FUNCTION_BLOCK FB_System_KKKW_145
VAR_INPUT

	Freigabe_auto			: BOOL;
	Freigabe_Deakt_auto		: BOOL;
	Betrieb_Anford_auto		: BOOL;

	Regelung_Modus_auto		: SINT;
	Regelung_Sollw_auto		: REAL;
END_VAR
VAR_OUTPUT
	{attribute 'OPC.UA.DA' := '1'}Parameter		: ST_System_KKKW_Parameter;   
	{attribute 'OPC.UA.DA' := '1'}Zustand			: ST_System_KKKW_Zustand;	
	{attribute 'OPC.UA.DA' := '1'}Stellwert		: ST_System_KKKW_Stellwert;  	
	{attribute 'OPC.UA.DA' := '1'}Steuerung		: ST_System_KKKW_Steuerung;  	
END_VAR
VAR
	Pumpe_145		: FB_PU;
	Stellventil_145	: FB_SV;
	Ablaufsteuerung	: FB_System_KKKW_Ablaufsteuerung;
	Logik			: FB_System_KKKW_Logik;
	Zustandscheck	: FB_System_KKKW_Zustandscheck;
	Stellwertscheck	: FB_System_KKKW_Stellwertscheck;
	Sollwertscheck	: FB_System_KKKW_Sollwertscheck;
END_VAR
VAR // added by the converter: edge detectors and wires of the graphical bodies
    _w1 : ANY;
END_VAR

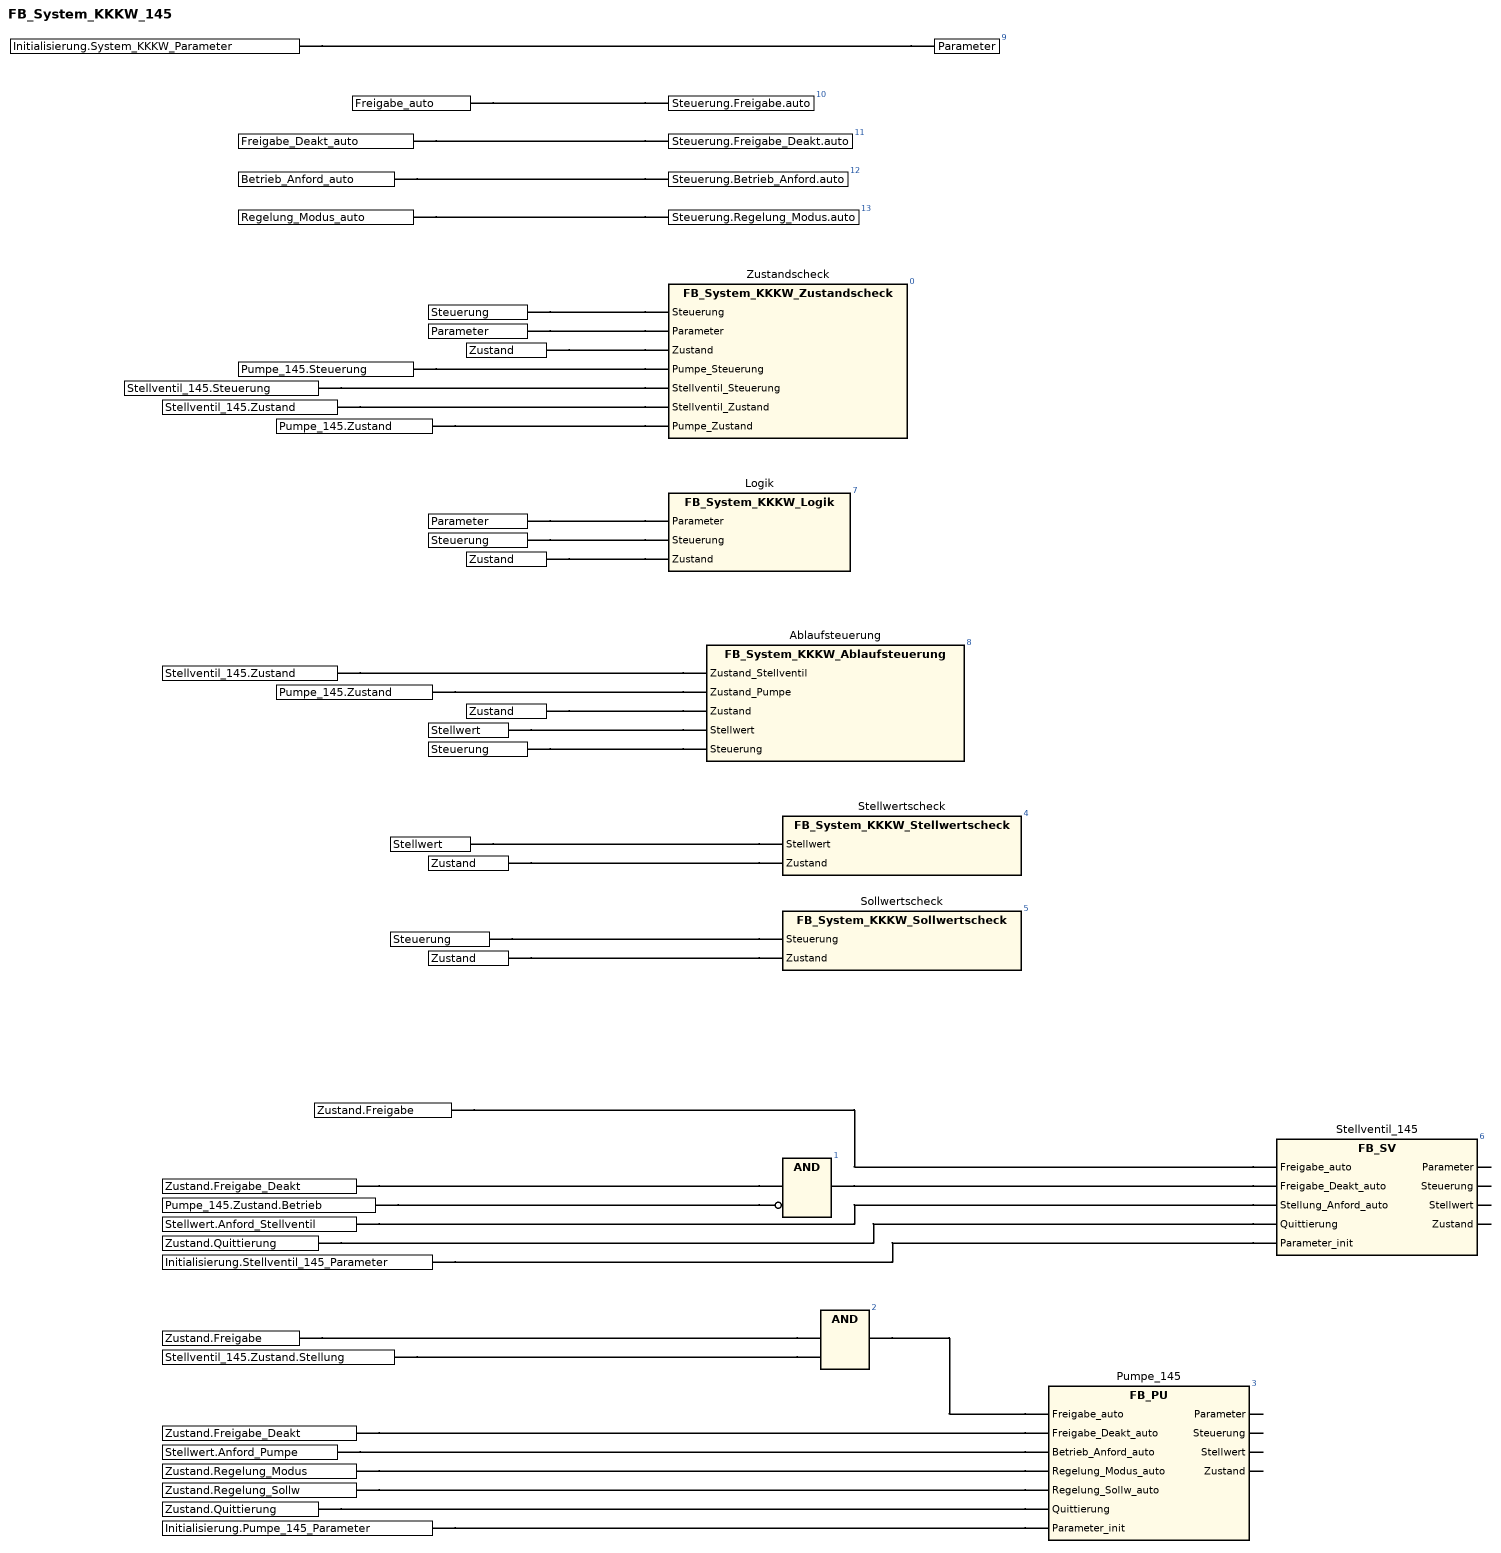
Zustandscheck(
    Steuerung := Steuerung,
    Parameter := Parameter,
    Zustand := Zustand,
    Pumpe_Steuerung := Pumpe_145.Steuerung,
    Stellventil_Steuerung := Stellventil_145.Steuerung,
    Stellventil_Zustand := Stellventil_145.Zustand,
    Pumpe_Zustand := Pumpe_145.Zustand); // FB_System_KKKW_Zustandscheck
_w1 := Zustand.Freigabe_Deakt AND NOT Pumpe_145.Zustand.Betrieb;
Pumpe_145(
    Freigabe_auto := Zustand.Freigabe AND Stellventil_145.Zustand.Stellung,
    Freigabe_Deakt_auto := Zustand.Freigabe_Deakt,
    Betrieb_Anford_auto := Stellwert.Anford_Pumpe,
    Regelung_Modus_auto := Zustand.Regelung_Modus,
    Regelung_Sollw_auto := Zustand.Regelung_Sollw,
    Quittierung := Zustand.Quittierung,
    Parameter_init := Initialisierung.Pumpe_145_Parameter); // FB_PU
Stellwertscheck(Stellwert := Stellwert, Zustand := Zustand); // FB_System_KKKW_Stellwertscheck
Sollwertscheck(Steuerung := Steuerung, Zustand := Zustand); // FB_System_KKKW_Sollwertscheck
Stellventil_145(
    Freigabe_auto := Zustand.Freigabe,
    Freigabe_Deakt_auto := _w1,
    Stellung_Anford_auto := Stellwert.Anford_Stellventil,
    Quittierung := Zustand.Quittierung,
    Parameter_init := Initialisierung.Stellventil_145_Parameter); // FB_SV
Logik(Parameter := Parameter, Steuerung := Steuerung, Zustand := Zustand); // FB_System_KKKW_Logik
Ablaufsteuerung(
    Zustand_Stellventil := Stellventil_145.Zustand,
    Zustand_Pumpe := Pumpe_145.Zustand,
    Zustand := Zustand,
    Stellwert := Stellwert,
    Steuerung := Steuerung); // FB_System_KKKW_Ablaufsteuerung
Parameter := Initialisierung.System_KKKW_Parameter;
Steuerung.Freigabe.auto := Freigabe_auto;
Steuerung.Freigabe_Deakt.auto := Freigabe_Deakt_auto;
Steuerung.Betrieb_Anford.auto := Betrieb_Anford_auto;
Steuerung.Regelung_Modus.auto := Regelung_Modus_auto;

END_FUNCTION_BLOCK

(* stored: Version 1.1.0.1, ProductVersion 3.1.4024.9
   POU FB_System_KKKW_145: Id {78722279-b58c-4fb5-a0ff-cce8874557a5}, SpecialFunc None *)
